// TIA Portal project "Hochregallager" (V14)

(* hardware
DEVICE "S7-1200-Station_1"  S7-1200 Station
   slot 0: "Baugruppenträger_0"  Rack  V1.0
   slot 1: "PLC"  CPU 1214C DC/DC/DC  6ES7 214-1AG40-0XB0  V4.1
   slot 3: "AQ 1x12BIT_1"  6ES7 232-4HA30-0XB0  V1.0
DEVICE "HMI"  KTP700 Basic PN
   slot 0: "HMI"  HMI  6AV2 123-2GB03-0AX0  13.0.1.0
   slot 1: "HMI_RT_1"  KTP700 Basic PN  6AV2 123-2GB03-0AX0  13.0.1.0
   slot 5: "HMI.IE_CP_1"  PROFINET Schnittstelle
      slot 1: "PROFINET Schnittstelle_1"  PROFINET Schnittstelle
         slot 1: "Port_1"  Port
*)

// ===== PLC "PLC"  CPU 1214C DC/DC/DC =====

VAR_GLOBAL   // PLC tag table "Standard-Variablentabelle"
   "System_Byte" AT %MB100 : Byte;
   "FirstScan" AT %M100.0 : Bool;
   "DiagStatusUpdate" AT %M100.1 : Bool;
   "AlwaysTRUE" AT %M100.2 : Bool;
   "AlwaysFALSE" AT %M100.3 : Bool;
   "Clock_Byte" AT %MB110 : Byte;
   "Clock_10Hz" AT %M110.0 : Bool;
   "Clock_5Hz" AT %M110.1 : Bool;
   "Clock_2.5Hz" AT %M110.2 : Bool;
   "Clock_2Hz" AT %M110.3 : Bool;
   "Clock_1.25Hz" AT %M110.4 : Bool;
   "Clock_1Hz" AT %M110.5 : Bool;
   "Clock_0.625Hz" AT %M110.6 : Bool;
   "Clock_0.5Hz" AT %M110.7 : Bool;
   "B1" AT %I0.0 : Bool;   // Werkstück/Palette auf Gabel
   "B2" AT %I0.1 : Bool;   // Gabel unten
   "B3" AT %I0.2 : Bool;   // Drehposition Links
   "B4" AT %I0.3 : Bool;   // Drehposition Rechts (Bedienpult)
   "B5" AT %I0.4 : Bool;   // Drehposition Mitte
   "B6" AT %I0.5 : Bool;   // Ebene Freigabe
   "Q1" AT %Q0.0 : Bool;   // Spindel-Motor abwärts
   "Q2" AT %Q0.1 : Bool;   // Spindel-Motor aufwärts
   "Q3" AT %Q0.2 : Bool;   // Drehmotor CW
   "Q4" AT %Q0.3 : Bool;   // Drehmotor CCW
   "AlleAusgänge" AT %QW0 : Word;
END_VAR

FUNCTION "fc_Hochregallager" : Void   // FC1, SCL
{ S7_Optimized_Access := 'TRUE' }
VERSION : 0.1
BEGIN
END_FUNCTION

ORGANIZATION_BLOCK "Main"   // OB1, LAD, ProgramCycle
TITLE = "Main Program Sweep (Cycle)"
{ S7_Optimized_Access := 'TRUE' }
VERSION : 0.1
   VAR_INPUT
      Initial_Call : Bool;   // Initial call of this OB
      Remanence : Bool;   // =True, if remanent data are available
   END_VAR
BEGIN

REGION Network 1: -Q1
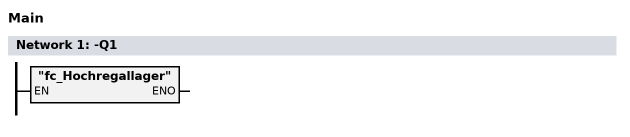
   RUNG wire#powerrail
      "fc_Hochregallager"()
   END_RUNG
   // the same network as SCL:
   "fc_Hochregallager"();
END_REGION
END_ORGANIZATION_BLOCK

ORGANIZATION_BLOCK "Startup"   // OB100, SCL, Startup
TITLE = "Complete Restart"
{ S7_Optimized_Access := 'TRUE' }
VERSION : 0.1
   VAR_INPUT
      LostRetentive : Bool;   // True if retentive data are lost
      LostRTC : Bool;   // True if date and time are lost
   END_VAR
BEGIN
   "AlleAusgänge" := 16#0000;
END_ORGANIZATION_BLOCK

(* ===== HMI "HMI_RT_1" =====
system functions are stored by id; their names below are inferred from use
connection "HMI_Verbindung_1": ETHERNET, SMART_S7_1200_OMS

HMI tags "Standard-Variablentabelle"
   "AlwaysTRUE" : Bool = PLC AlwaysTRUE AT %M100.2, 100 ms
   "Q1" : Bool = PLC Q1 AT %Q0.0, 100 ms
   "Q2" : Bool = PLC Q2 AT %Q0.1, 100 ms
   "Q3" : Bool = PLC Q3 AT %Q0.2, 100 ms
   "Q4" : Bool = PLC Q4 AT %Q0.3, 100 ms
   "B1" : Bool = PLC B1 AT %I0.0, 100 ms
   "B2" : Bool = PLC B2 AT %I0.1, 100 ms
   "B3" : Bool = PLC B3 AT %I0.2, 100 ms
   "B4" : Bool = PLC B4 AT %I0.3, 100 ms
   "B5" : Bool = PLC B5 AT %I0.4, 100 ms
   "B6" : Bool = PLC B6 AT %I0.5, 100 ms

screen "Hochregallager" 800x480
   TextField "Textfeld_2" at 279,5 size 250x43; Text 'Hochregallager'
   Button "Schaltfläche_1" at 655,65 size 80x40; TextOff 'Auf'; TextOn 'Start'
      on Press: SetBit("Q1")
      on Release: ResetBit("Q1")
   Circle "Kreis_3" at 60,110 size 50x50
      Appearance <- "B2"
   TextField "Textfeld_4" at 110,125 size 104x23; Text 'Gabel unten'
   Circle "Kreis_5" at 60,60 size 50x50
      Appearance <- "B1"
   TextField "Textfeld_6" at 110,75 size 243x23; Text 'Werkstück/Palette auf Gabel'
   Circle "Kreis_1" at 60,160 size 50x50
      Appearance <- "B3"
   Circle "Kreis_2" at 60,210 size 50x50
      Appearance <- "B4"
   TextField "Textfeld_1" at 110,175 size 156x23; Text 'Drehposition Links'
   TextField "Textfeld_3" at 110,225 size 276x23; Text 'Drehposition Rechts (Bedienpult)'
   Button "Schaltfläche_2" at 665,160 size 80x40; TextOn 'Start'; TextOff 'Ab'
      on Release: ResetBit("Q2")
      on Press: SetBit("Q2")
   Button "Schaltfläche_3" at 600,115 size 80x40; TextOn 'Start'; TextOff 'CW'
      on Release: ResetBit("Q3")
      on Press: SetBit("Q3")
   Button "Schaltfläche_4" at 710,115 size 80x40; TextOn 'Start'; TextOff 'CCW'
      on Release: ResetBit("Q4")
      on Press: SetBit("Q4")
   TextField "Textfeld_5" at 110,275 size 157x23; Text 'Drehposition Mitte'
   TextField "Textfeld_7" at 110,320 size 131x23; Text 'Ebene Freigabe'
   Circle "Kreis_4" at 60,260 size 50x50
      Appearance <- "B5"
   Circle "Kreis_6" at 60,310 size 50x50
      Appearance <- "B6"
*)